INTERFACE I_ObjectRunner

METHOD AddComponent : HRESULT
VAR_INPUT
	CyclicModule : ICyclic;
END_VAR
END_METHOD

END_INTERFACE

(* stored: Version 1.1.0.1, ProductVersion 3.1.4024.12
   Itf I_ObjectRunner: Id {7ae64750-6a2f-446f-b3b5-fa2d9501c423}
   Method AddComponent: Id {119d0526-b150-47f1-ab98-856e052618fb} *)
